PROGRAM DIGI_Main
VAR

//	IPAdress		: STRING 	:= '192.168.1.132';
//	Port			: UINT		:= 5000;
	IPAddress		: STRING 	:= '10.0.110.19';
	Port			: UINT		:= 6060;
	UpdatePeriod	: TIME		:= T#60S;
	Timer 			: BOOL;
	
	sAPI_addr		: STRING := '/upload?file=SIM_ASRSAction.json';
	API_MSG			: STRING(3500);
	HttpSend		: BOOL := FALSE;
	bSuccess		: BOOL;
	bError			: BOOL;
	
	fb_TimeStamp	: FB_UpdateTimeStamp_1;
	fb_httppost		: FB_EventHTTP_Post;
	fbTON 	: TON;
	fbTOFF 	: TON;
	Rise1	: R_TRIG;
	
	fbHttpProcess	: FB_IotHttpClient :=(	sHostName			:= IPAddress,
								  			bKeepAlive			:= TRUE, 
											tConnectionTimeout	:= T#10S);
	enabler	: BOOL;	
	
	//rising edges
	rHome	:	R_TRIG;
	rToWait	:	R_TRIG;
	fToWait	:	F_TRIG;
	rPick	:	R_TRIG;
	fPick	:	F_TRIG;
	fPlace01	:	F_TRIG;
	fPlace02	:	F_TRIG;
	fPlace03	:	F_TRIG;
	fPlace04	:	F_TRIG;
	fPlace05	:	F_TRIG;
	fPlace06	:	F_TRIG;
	fPlace07	:	F_TRIG;
	fPlace08	:	F_TRIG;
	fPlace09	:	F_TRIG;
	fPlace10	:	F_TRIG;
	fPlace11	:	F_TRIG;
	fPlace12	:	F_TRIG;
	fPlace13	:	F_TRIG;
	fPlace14	:	F_TRIG;
	fPlace15	:	F_TRIG;
	fPlace16	:	F_TRIG;
	fPlace17	:	F_TRIG;
	fPlace18	:	F_TRIG;
	
//	rHome	:	R_TRIG;
//	rToWait	:	R_TRIG;
//	rPick	:	R_TRIG;
//	fPlace01	:	F_TRIG;
//	rPlace02	:	R_TRIG;
//	rPlace03	:	R_TRIG;
//	rPlace04	:	R_TRIG;
//	rPlace05	:	R_TRIG;
//	rPlace06	:	R_TRIG;
//	rPlace07	:	R_TRIG;
//	rPlace08	:	R_TRIG;
//	rPlace09	:	R_TRIG;
//	rPlace10	:	R_TRIG;
//	rPlace11	:	R_TRIG;
//	rPlace12	:	R_TRIG;
//	rPlace13	:	R_TRIG;
//	rPlace14	:	R_TRIG;
//	rPlace15	:	R_TRIG;
//	rPlace16	:	R_TRIG;
//	rPlace17	:	R_TRIG;
//	rPlace18	:	R_TRIG;
	
	
	
END_VAR


IF NOT fbHttpProcess.bConfigured THEN 
	fbHttpProcess.nHostPort 				:= Port;
	fbHttpProcess.stTLS.bNoServerCertCheck 	:= FALSE;
END_IF
	
fb_TimeStamp();

rHome(CLK := IO_KUKA.bGo_home_InProcess);
rToWait(CLK := IO_KUKA.bStandby_pos_InProcess);
//fToWait(CLK := IO_KUKA.bRA_pos1_InProcess OR IO_KUKA.bRA_pos2_InProcess );
rPick(CLK := IO_KUKA.bBin_pickup_InProcess);


fPlace01(CLK := IO_control.bRA_pos1);
fPlace02(CLK := IO_control.bRA_pos2);
fPlace03(CLK := IO_control.bRA_pos3);
fPlace04(CLK := IO_control.bRA_pos4);
fPlace05(CLK := IO_control.bRA_pos5);
fPlace06(CLK := IO_control.bRA_pos6);
fPlace07(CLK := IO_control.bRB_pos7);
fPlace08(CLK := IO_control.bRB_pos8);
fPlace09(CLK := IO_control.bRB_pos9);
fPlace10(CLK := IO_control.bRB_pos10);
fPlace11(CLK := IO_control.bRB_pos11);
fPlace12(CLK := IO_control.bRB_pos12);
fPlace13(CLK := IO_control.bRC_pos13);
fPlace14(CLK := IO_control.bRC_pos14);
fPlace15(CLK := IO_control.bRC_pos15);
fPlace16(CLK := IO_control.bRC_pos16);
fPlace17(CLK := IO_control.bRC_pos17);
fPlace18(CLK := IO_control.bRC_pos18);

Rise1(CLK:= enabler);

IF fb_TimeStamp.timeValid THEN
	IF Rise1.Q THEN
		IO.sActionkey := 'Testing';
		IO.iActionval := 1;
		DIGIIOT_UPDATE(SystemTime := fb_TimeStamp.timestampSeconds);
		HttpSend := TRUE;
	END_IF
	
//	IF rHome.Q THEN
//		IO.sActionkey := 'Home';
//		IO.iActionval := 1;
//		DIGIIOT_UPDATE(SystemTime := fb_TimeStamp.timestampSeconds);
//		HttpSend := TRUE;
//	END_IF
	
	IF rToWait.Q THEN
		IO.sActionkey := 'ToWait';
		IO.iActionval := 1;
		DIGIIOT_UPDATE(SystemTime := fb_TimeStamp.timestampSeconds);
		HttpSend := TRUE;
	END_IF
	
	IF rPick.Q THEN
		IO.sActionkey := 'BinPickUp';
		IO.iActionval := 1;
		DIGIIOT_UPDATE(SystemTime := fb_TimeStamp.timestampSeconds);
		HttpSend := TRUE;
	END_IF
	
	IF fPlace01.Q THEN
		IO.sActionkey := 'BinPlace_01';
		IO.iActionval := 1;
		DIGIIOT_UPDATE(SystemTime := fb_TimeStamp.timestampSeconds);
		HttpSend := TRUE;
	END_IF
	
	IF fPlace02.Q THEN
		IO.sActionkey := 'BinPlace_02';
		IO.iActionval := 1;
		DIGIIOT_UPDATE(SystemTime := fb_TimeStamp.timestampSeconds);
		HttpSend := TRUE;
	END_IF
	
	IF fPlace03.Q THEN
		IO.sActionkey := 'BinPlace_03';
		IO.iActionval := 1;
		DIGIIOT_UPDATE(SystemTime := fb_TimeStamp.timestampSeconds);
		HttpSend := TRUE;
	END_IF
	
	IF fPlace04.Q THEN
		IO.sActionkey := 'BinPlace_04';
		IO.iActionval := 1;
		DIGIIOT_UPDATE(SystemTime := fb_TimeStamp.timestampSeconds);
		HttpSend := TRUE;
	END_IF
	
	IF fPlace05.Q THEN
		IO.sActionkey := 'BinPlace_05';
		IO.iActionval := 1;
		DIGIIOT_UPDATE(SystemTime := fb_TimeStamp.timestampSeconds);
		HttpSend := TRUE;
	END_IF
	
	IF fPlace06.Q THEN
		IO.sActionkey := 'BinPlace_06';
		IO.iActionval := 1;
		DIGIIOT_UPDATE(SystemTime := fb_TimeStamp.timestampSeconds);
		HttpSend := TRUE;
	END_IF
	
	IF fPlace07.Q THEN
		IO.sActionkey := 'BinPlace_07';
		IO.iActionval := 1;
		DIGIIOT_UPDATE(SystemTime := fb_TimeStamp.timestampSeconds);
		HttpSend := TRUE;
	END_IF
	
	IF fPlace08.Q THEN
		IO.sActionkey := 'BinPlace_08';
		IO.iActionval := 1;
		DIGIIOT_UPDATE(SystemTime := fb_TimeStamp.timestampSeconds);
		HttpSend := TRUE;
	END_IF
	
	IF fPlace09.Q THEN
		IO.sActionkey := 'BinPlace_09';
		IO.iActionval := 1;
		DIGIIOT_UPDATE(SystemTime := fb_TimeStamp.timestampSeconds);
		HttpSend := TRUE;
	END_IF
	
	IF fPlace10.Q THEN
		IO.sActionkey := 'BinPlace_10';
		IO.iActionval := 1;
		DIGIIOT_UPDATE(SystemTime := fb_TimeStamp.timestampSeconds);
		HttpSend := TRUE;
	END_IF
	
	IF fPlace11.Q THEN
		IO.sActionkey := 'BinPlace_11';
		IO.iActionval := 1;
		DIGIIOT_UPDATE(SystemTime := fb_TimeStamp.timestampSeconds);
		HttpSend := TRUE;
	END_IF
	
	IF fPlace12.Q THEN
		IO.sActionkey := 'BinPlace_12';
		IO.iActionval := 1;
		DIGIIOT_UPDATE(SystemTime := fb_TimeStamp.timestampSeconds);
		HttpSend := TRUE;
	END_IF
	
	IF fPlace13.Q THEN
		IO.sActionkey := 'BinPlace_13';
		IO.iActionval := 1;
		DIGIIOT_UPDATE(SystemTime := fb_TimeStamp.timestampSeconds);
		HttpSend := TRUE;
	END_IF
	
	IF fPlace14.Q THEN
		IO.sActionkey := 'BinPlace_14';
		IO.iActionval := 1;
		DIGIIOT_UPDATE(SystemTime := fb_TimeStamp.timestampSeconds);
		HttpSend := TRUE;
	END_IF
	
	IF fPlace15.Q THEN
		IO.sActionkey := 'BinPlace_15';
		IO.iActionval := 1;
		DIGIIOT_UPDATE(SystemTime := fb_TimeStamp.timestampSeconds);
		HttpSend := TRUE;
	END_IF
	
	IF fPlace16.Q THEN
		IO.sActionkey := 'BinPlace_16';
		IO.iActionval := 1;
		DIGIIOT_UPDATE(SystemTime := fb_TimeStamp.timestampSeconds);
		HttpSend := TRUE;
	END_IF
	
	IF fPlace17.Q THEN
		IO.sActionkey := 'BinPlace_17';
		IO.iActionval := 1;
		DIGIIOT_UPDATE(SystemTime := fb_TimeStamp.timestampSeconds);
		HttpSend := TRUE;
	END_IF
	
	IF fPlace18.Q THEN
		IO.sActionkey := 'BinPlace_18';
		IO.iActionval := 1;
		DIGIIOT_UPDATE(SystemTime := fb_TimeStamp.timestampSeconds);
		HttpSend := TRUE;
	END_IF
	
	IF fbHttpProcess.bConfigured THEN 
		fb_httppost( 	bSend		:= HttpSend, 
						fbClient	:= fbHttpProcess, 
						API_URI		:= sAPI_addr,
						API_Msg		:= IO.DIGI_MSG,
						bSuccess 	=> bSuccess,
						bError		=> bError );
						
		IF fb_httppost.bSuccess OR fb_httppost.bError THEN
			HttpSend := FALSE;
		END_IF
	END_IF 
	fbHttpProcess.Execute();
END_IF






//IF fb_TimeStamp.timeValid THEN
		
//	Rise1(CLK:= enabler);
//	IF Rise1.Q THEN
//		HttpSend := TRUE;
//		DIGIIOT_UPDATE(SystemTime := fb_TimeStamp.timestampSeconds);
//	END_IF

//	IF fbHttpProcess.bConfigured THEN 
//		fb_httppost( 	bSend		:= HttpSend, 
//						fbClient	:= fbHttpProcess, 
//						API_URI		:= '/upload',
//						API_Msg		:= IO.DIGI_MSG,
//						bSuccess 	=> bSuccess,
//						bError		=> bError );
						
//		IF fb_httppost.bSuccess OR fb_httppost.bError THEN
//			HttpSend := FALSE;
//		END_IF
//	END_IF 
//	fbHttpProcess.Execute();
//END_IF

END_PROGRAM

(* stored: Version 1.1.0.1, ProductVersion 3.1.4024.12
   POU DIGI_Main: Id {bc02980f-fea0-4e7e-8235-d2e7da73e07d}, SpecialFunc None *)
